FUNCTION_BLOCK Backout
VAR_INPUT
	Backout_switch:BOOL;
	Reset:BOOL;
	Left_overwind:BOOL;
	Left_underwind:BOOL;
	Right_overwind:BOOL;
	Right_underwind:BOOL;
	Brake_lever_on:BOOL;
	Lever_neutral:BOOL;
	Fwd:BOOL;
	Rev:BOOL;
	Forward_backout_relay_fb:BOOL;
	Reverse_backout_relay_fb:BOOL;
END_VAR
VAR_OUTPUT
	Forward_backout_relay:BOOL;
	Reverse_backout_relay:BOOL;
	Forward_xcheck_fault:BOOL;
	Reverse_xcheck_fault:BOOL;
END_VAR
VAR
	Bor_set1:BOOL;
	Bor_set2:BOOL;
	Bor_set3:BOOL;
	Bor_set4:BOOL;
	Bor_rst1:BOOL;
	Bor_rst2:BOOL;
	Bor_rst3:BOOL;
	Bor_rst4:BOOL;
	Bor_rst5:BOOL;
	RS_0: RS;
	TON_0: TON;
	F_TRIG_0: F_TRIG;
END_VAR

Backout_main();

METHOD Backout_main
VAR_INPUT
END_VAR
VAR_INST // added by the converter: edge detectors and wires of the graphical bodies
    _w1, _w4, _w5, _w7 : BOOL;
    _w2, _w3, _w6 : ANY;
END_VAR
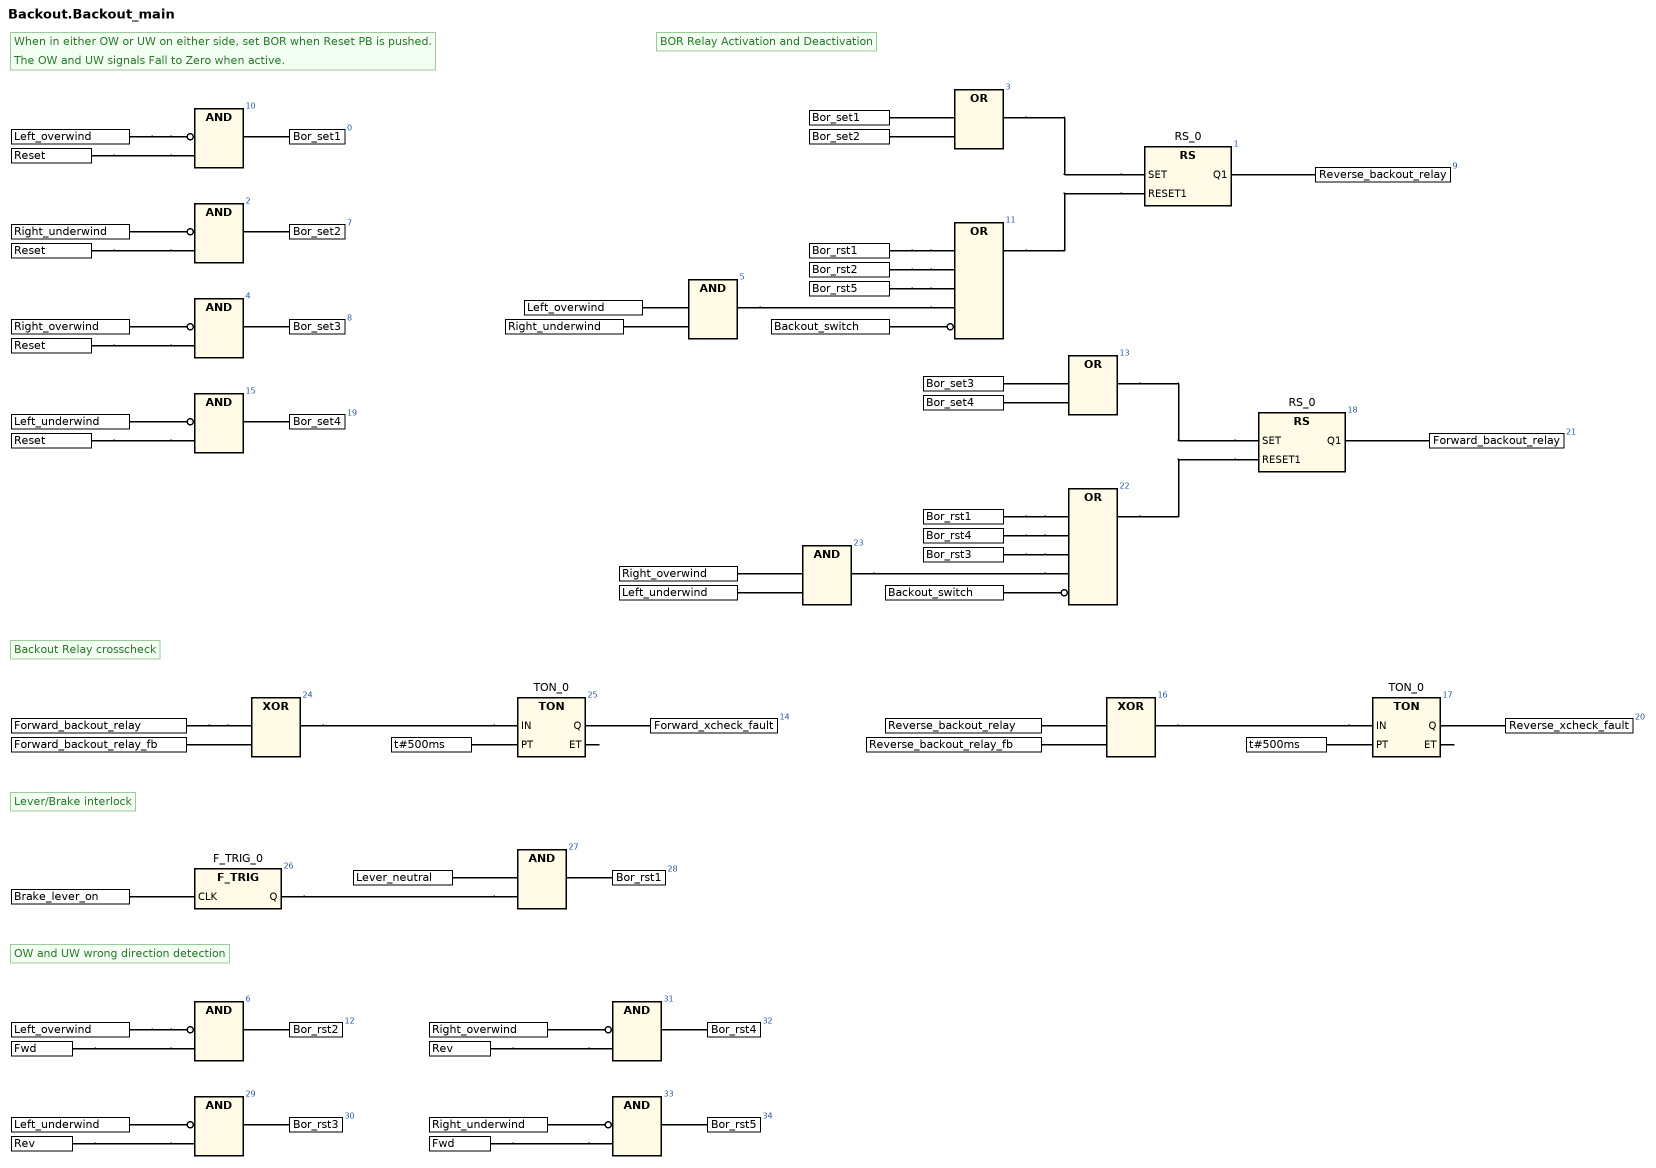
Bor_set1 := _w1;
RS_0(SET := _w2, RESET1 := _w3); // RS
// BOR Relay Activation and Deactivation
_w2 := Bor_set1 OR Bor_set2;
// OW and UW wrong direction detection
Bor_set2 := NOT Right_underwind AND Reset;
Bor_set3 := NOT Right_overwind AND Reset;
Reverse_backout_relay := RS_0.Q1;
// When in either OW or UW on either side, set BOR when Reset PB is pushed.
// The OW and UW signals Fall to Zero when active.
_w1 := NOT Left_overwind AND Reset;
_w3 := Bor_rst1 OR Bor_rst2 OR Bor_rst5 OR Left_overwind AND Right_underwind OR NOT Backout_switch;
Bor_rst2 := NOT Left_overwind AND Fwd;
_w4 := Bor_set3 OR Bor_set4;
Forward_xcheck_fault := TON_0.Q;
_w5 := NOT Left_underwind AND Reset;
TON_0(IN := Reverse_backout_relay XOR Reverse_backout_relay_fb, PT := t#500ms); // TON
RS_0(SET := _w4, RESET1 := _w6); // RS
Bor_set4 := _w5;
Reverse_xcheck_fault := TON_0.Q;
Forward_backout_relay := RS_0.Q1;
_w6 := Bor_rst1 OR Bor_rst4 OR Bor_rst3 OR _w7 OR NOT Backout_switch;
_w7 := Right_overwind AND Left_underwind;
// Backout Relay crosscheck
TON_0(IN := Forward_backout_relay XOR Forward_backout_relay_fb, PT := t#500ms); // TON
// Lever/Brake interlock
F_TRIG_0(CLK := Brake_lever_on); // F_TRIG
Bor_rst1 := Lever_neutral AND F_TRIG_0.Q;
Bor_rst3 := NOT Left_underwind AND Rev;
Bor_rst4 := NOT Right_overwind AND Rev;
Bor_rst5 := NOT Right_underwind AND Fwd;
END_METHOD

END_FUNCTION_BLOCK

(* stored: Version 1.1.0.1, ProductVersion 3.1.4024.0
   POU Backout: Id {9a5fecb9-7ff1-4f14-bf3a-a287dd5735fd}, SpecialFunc None
   Method Backout_main: Id {6617efd7-da41-4b37-a8f0-683ab38bd9c5} *)
